ADAPTER RegisterServiceAdp (* Register Service Adapter *)
  (* Standard: 61499-2; Description: Copyright (c) 2018 fortiss GmbH This program and the accompanying materials are made available under the terms of the Eclipse Public License 2.0 which is available at https://www.eclipse.org/legal/epl-2.0/ SPDX-License-Identifier: EPL-2.0 *)
  (* Version 1.0, 2018-09-21, Jose Cabral, fortiss GmbH *)
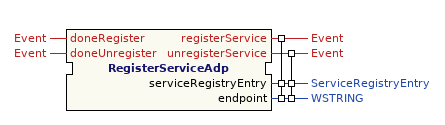
  EVENT_INPUT
    doneRegister; (* Register finished *)
    doneUnregister; (* Unregister finished *)
  END_EVENT
  EVENT_OUTPUT
    registerService WITH serviceRegistryEntry, endpoint; (* Register the services *)
    unregisterService WITH serviceRegistryEntry, endpoint; (* Unregister the service *)
  END_EVENT
  VAR_OUTPUT
    serviceRegistryEntry : ServiceRegistryEntry; (* Service Registry Entry for register or unregister *)
    endpoint : WSTRING; (* Endpoint (IP:PORT/URI) of the Service Registry (not officially in the documentation, but it simplifies the FBs) *)
  END_VAR
  (* Service SOCKET/PLUG: Register Service Adapter *)
END_ADAPTER
